Staubli VAL3: OnF2.pgx

program OnF2()
  local num l_ni
  local bool l_bRes
begin
  switch nPage
    case 0
      //模拟
      call SimuMain()
    break
    case 1
      //insert
      nSelected=nSelected+1
      insert(prd:pDemo[nSelected])
      prd:pDemo[nSelected]=here(Tool:tTool[prd:sToolName],Frame:fFrame[prd:sFrameName])
      insert(prd:sPtParameter[nSelected])
      //添加点的信息
    break
    case 2
    break
    case 3
    break
    case 4
    break

  endSwitch

end
